{attribute addProperty BoxType "EP4378-1022-0017"}
{attribute addProperty Id "StatusAT %I*Status_845218981621ValueAT %I*INT16217"}
{attribute addProperty CRC "142569927"}
{attribute addProperty SizeInBites "32"}
{attribute addProperty SizeInBytes "4"}
TYPE AI_X05_Pin2_Standard_087F71C7 :
STRUCT
	{attribute addProperty Name "Status"}
	Status AT %I* : Status_84521898;
	{attribute addProperty Name "Value"}
	Value AT %I* : INT;
END_STRUCT
END_TYPE

(* stored: Version 1.2.0.0, ProductVersion 3.1.4024.9
   DUT AI_X05_Pin2_Standard_087F71C7: Id {58c4fc68-8029-4ee9-8558-0ecee8bb1d8f} *)
